INTERFACE PUBLIC I_ExecuteCommands

METHOD PUBLIC Abort
END_METHOD

METHOD PUBLIC Hold
END_METHOD

METHOD PUBLIC StateComplete
END_METHOD

METHOD PUBLIC Stop
END_METHOD

METHOD PUBLIC Suspend
END_METHOD

END_INTERFACE

(* stored: Version 1.1.0.1, ProductVersion 3.1.4026.6
   Itf I_ExecuteCommands: Id {9dab06e0-c06a-0aec-34db-a51978aa62c9}
   Method Abort: Id {a61a6c0b-6030-4475-b992-98b2b130c10d}
   Method Hold: Id {e0475413-9d6e-0d10-1b86-688b115f827f}
   Method StateComplete: Id {243d399f-34e0-4999-a92c-fac012d19dfe}
   Method Stop: Id {de296dca-ddbe-413c-a5ef-5e88b622c2cf}
   Method Suspend: Id {2f703afa-fea1-0aae-04b9-1ccf0ad65f2e} *)
